// Mitsubishi GX Works2 project: servo_teach_blockloop   PLC: Q02/Q02H

PROGRAM MAIN
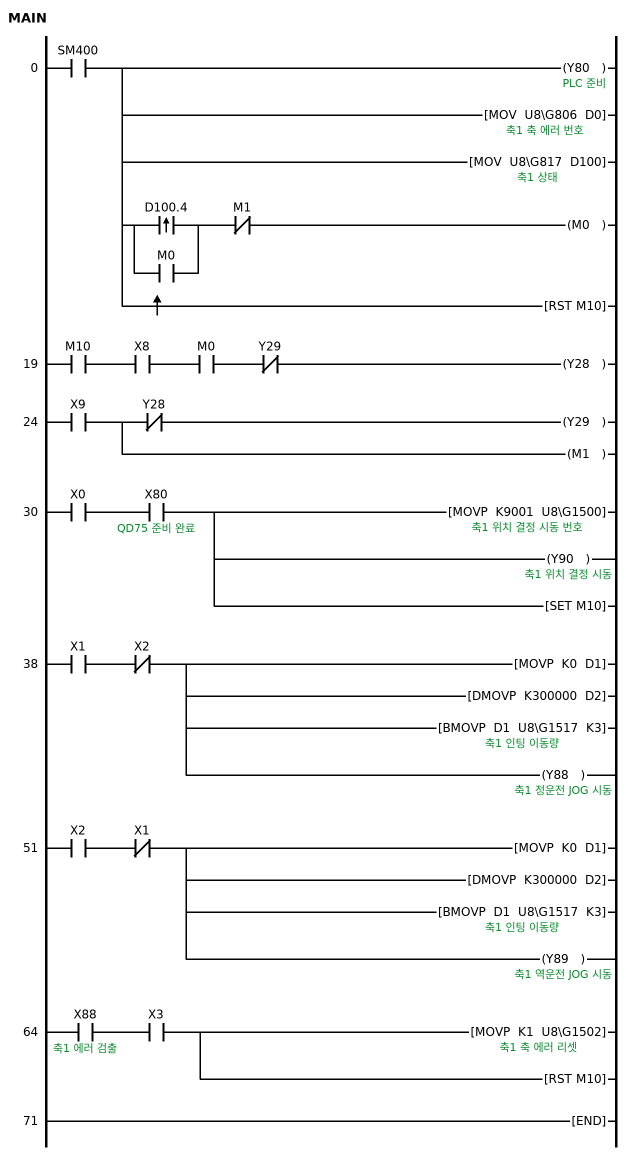
0     LD      SM400
      OUT     Y80  ; PLC 준비
      MOV     U8\G806 D0  ; 축1 축 에러 번호
      MOV     U8\G817 D100  ; 축1 상태
      MPS
      LDP     D100.4
      OR      M0
      ANB
      ANI     M1
      OUT     M0
      MPP
      MEP
      RST     M10
19    LD      M10
      AND     X8
      AND     M0
      ANI     Y29
      OUT     Y28
24    LD      X9
      MPS
      ANI     Y28
      OUT     Y29
      MPP
      OUT     M1
30    LD      X0
      AND     X80  ; QD75 준비 완료
      MOVP    K9001 U8\G1500  ; 축1 위치 결정 시동 번호
      OUT     Y90  ; 축1 위치 결정 시동
      SET     M10
38    LD      X1
      ANI     X2
      MOVP    K0 D1
      DMOVP   K300000 D2
      BMOVP   D1 U8\G1517 K3  ; 축1 인팅 이동량
      OUT     Y88  ; 축1 정운전 JOG 시동
51    LD      X2
      ANI     X1
      MOVP    K0 D1
      DMOVP   K300000 D2
      BMOVP   D1 U8\G1517 K3
      OUT     Y89  ; 축1 역운전 JOG 시동
64    LD      X88  ; 축1 에러 검출
      AND     X3
      MOVP    K1 U8\G1502  ; 축1 축 에러 리셋
      RST     M10
71    END
END_PROGRAM

PROGRAM MAIN1
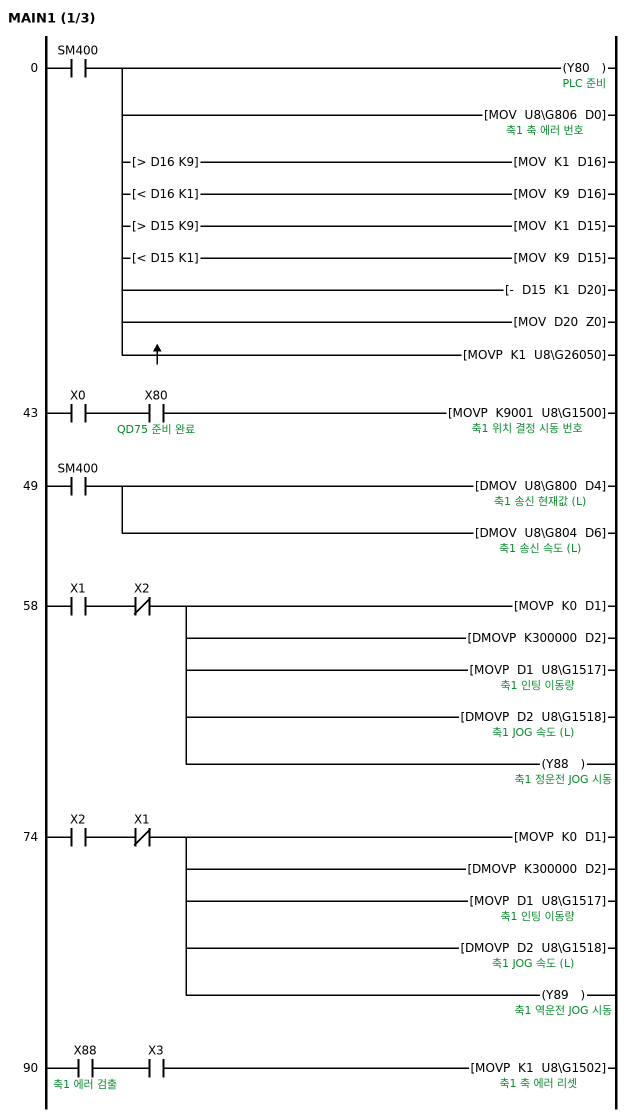
0     LD      SM400
      OUT     Y80  ; PLC 준비
      MOV     U8\G806 D0  ; 축1 축 에러 번호
      MPS
      AND>    D16 K9
      MOV     K1 D16
      MRD
      AND<    D16 K1
      MOV     K9 D16
      MRD
      AND>    D15 K9
      MOV     K1 D15
      MRD
      AND<    D15 K1
      MOV     K9 D15
      MPP
      -       D15 K1 D20
      MOV     D20 Z0
      MEP
      MOVP    K1 U8\G26050
43    LD      X0
      AND     X80  ; QD75 준비 완료
      MOVP    K9001 U8\G1500  ; 축1 위치 결정 시동 번호
49    LD      SM400
      DMOV    U8\G800 D4  ; 축1 송신 현재값 (L)
      DMOV    U8\G804 D6  ; 축1 송신 속도 (L)
58    LD      X1
      ANI     X2
      MOVP    K0 D1
      DMOVP   K300000 D2
      MOVP    D1 U8\G1517  ; 축1 인팅 이동량
      DMOVP   D2 U8\G1518  ; 축1 JOG 속도 (L)
      OUT     Y88  ; 축1 정운전 JOG 시동
74    LD      X2
      ANI     X1
      MOVP    K0 D1
      DMOVP   K300000 D2
      MOVP    D1 U8\G1517
      DMOVP   D2 U8\G1518
      OUT     Y89  ; 축1 역운전 JOG 시동
90    LD      X88  ; 축1 에러 검출
      AND     X3
      MOVP    K1 U8\G1502  ; 축1 축 에러 리셋
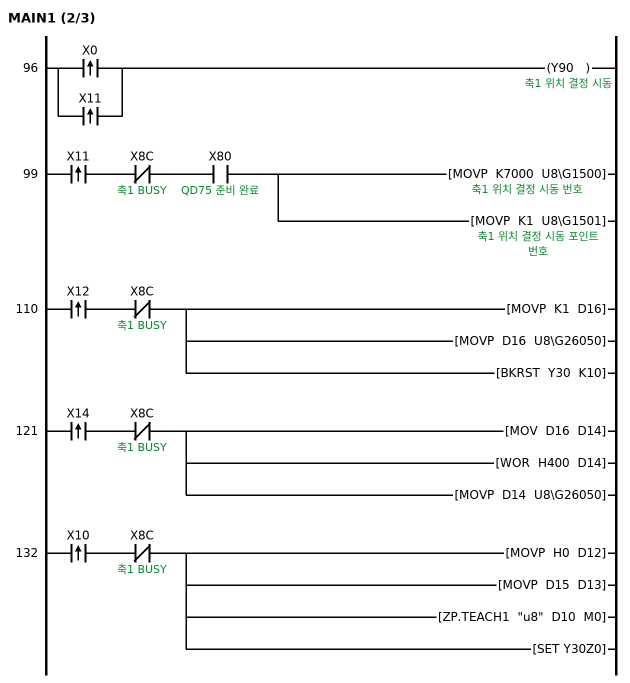
96    LDP     X0
      ORP     X11
      OUT     Y90  ; 축1 위치 결정 시동
99    LDP     X11
      ANI     X8C  ; 축1 BUSY
      AND     X80  ; QD75 준비 완료
      MOVP    K7000 U8\G1500
      MOVP    K1 U8\G1501  ; 축1 위치 결정 시동 포인트 번호
110   LDP     X12
      ANI     X8C  ; 축1 BUSY
      MOVP    K1 D16
      MOVP    D16 U8\G26050
      BKRST   Y30 K10
121   LDP     X14
      ANI     X8C  ; 축1 BUSY
      MOV     D16 D14
      WOR     H400 D14
      MOVP    D14 U8\G26050
132   LDP     X10
      ANI     X8C  ; 축1 BUSY
      MOVP    H0 D12
      MOVP    D15 D13
      ZP.TEACH1 "u8" D10 M0
      SET     Y30Z0
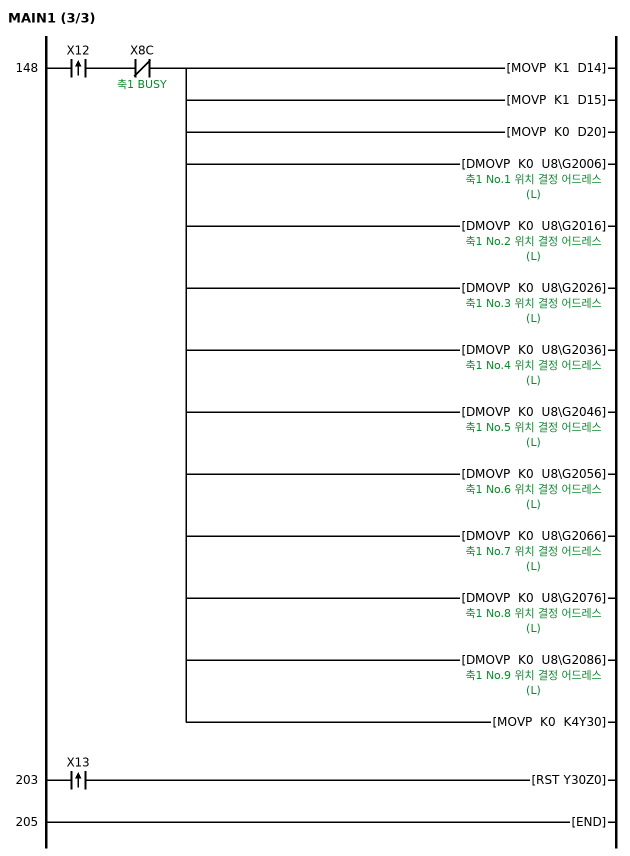
148   LDP     X12
      ANI     X8C  ; 축1 BUSY
      MOVP    K1 D14
      MOVP    K1 D15
      MOVP    K0 D20
      DMOVP   K0 U8\G2006  ; 축1 No.1 위치 결정 어드레스 (L)
      DMOVP   K0 U8\G2016  ; 축1 No.2 위치 결정 어드레스 (L)
      DMOVP   K0 U8\G2026  ; 축1 No.3 위치 결정 어드레스 (L)
      DMOVP   K0 U8\G2036  ; 축1 No.4 위치 결정 어드레스 (L)
      DMOVP   K0 U8\G2046  ; 축1 No.5 위치 결정 어드레스 (L)
      DMOVP   K0 U8\G2056  ; 축1 No.6 위치 결정 어드레스 (L)
      DMOVP   K0 U8\G2066  ; 축1 No.7 위치 결정 어드레스 (L)
      DMOVP   K0 U8\G2076  ; 축1 No.8 위치 결정 어드레스 (L)
      DMOVP   K0 U8\G2086  ; 축1 No.9 위치 결정 어드레스 (L)
      MOVP    K0 K4Y30
203   LDP     X13
      RST     Y30Z0
205   END
END_PROGRAM

// device comments not shown above
X81  ; 동기용 플래그
X84  ; 축1 M 코드 ON
X85  ; 축2 M 코드 ON
X89  ; 축2 에러 검출
X8D  ; 축2 BUSY
X90  ; 축1 시동 완료
X91  ; 축2 시동 완료
X94  ; 축1 위치 결정 완료
X95  ; 축2 위치 결정 완료
Y84  ; 축1 축 정지
Y85  ; 축2 축 정지
Y8A  ; 축2 정운전 JOG 시동
Y8B  ; 축2 역운전 JOG 시동
Y91  ; 축2 위치 결정 시동
Y94  ; 축1 실행 금지 플래그
Y95  ; 축2 실행 금지 플래그
